{attribute addProperty BoxType "ELX3181-0000-0016"}
{attribute addProperty Id "Ch_1Ch_1_9A58320E3240WcStateAT %I*WcState_98A4DF7520.250InfoDataAT %I*InfoData_275E3363128160"}
{attribute addProperty CRC "3569457747"}
{attribute addProperty SizeInBites "162"}
{attribute addProperty SizeInBytes "20.25"}
TYPE ELX3181_644058BD :
STRUCT
	{attribute addProperty Name "Ch_1"}
	Ch_1 : Ch_1_9A58320E;
	{attribute addProperty Name "WcState"}
	WcState : WcState_98A4DF75;
	{attribute addProperty Name "InfoData"}
	InfoData : InfoData_275E3363;
END_STRUCT
END_TYPE

(* stored: Version 1.2.0.0, ProductVersion 3.1.4024.9
   DUT ELX3181_644058BD: Id {a32577cb-d643-413e-96ac-4f88542ba128} *)
